FUNCTION_BLOCK Q_StringValue (* Command Change String Value ( Part 6 - F.24 ) *)
  (* Standard: ISO 11783-6; Description: This command sends a string to the VT. The length of the string including '\0' may not be longer than the define ISO_VTC_CMD_STR_MAX_LENGTH. Take care that '\0' is trailed. Return values iso_s16 - E_NO_ERR - transport started - E_OVERFLOW - buffer overflow - E_NOACT - Command not possible in current state - E_NO_INSTANCE - No VT client available *)
  (* Version 1.0, 2022-07-08, franz *)
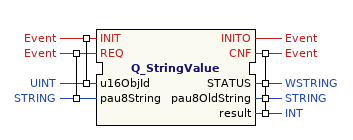
  EVENT_INPUT
    INIT WITH u16ObjId; (* Service Initialization *)
    REQ WITH pau8String; (* Service Request *)
  END_EVENT
  EVENT_OUTPUT
    INITO; (* Initialization Confirm *)
    CNF WITH STATUS, pau8OldString, result; (* Confirmation of Requested Service *)
  END_EVENT
  VAR_INPUT
    u16ObjId : UINT; (* Object ID *)
    pau8String : STRING; (* Pointer to string *)
  END_VAR
  VAR_OUTPUT
    STATUS : WSTRING; (* Service Status *)
    pau8OldString : STRING; (* Old pointer to string *)
    result : INT; (* retval see description *)
  END_VAR
END_FUNCTION_BLOCK
